PROGRAM AntiBlockingDamper
VAR
	fbHVACAntiBlockingDamper: FB_HVACAntiBlockingDamper;
	eDataSecurityType: E_HVACDataSecurityType := E_HVACDataSecurityType.eHVACDataSecurityType_Idle;
	bSetDefault: BOOL;
	bEnable: BOOL;
	bDisable: BOOL;
	ryDamper: REAL;
	dtSystemTime: DATE_AND_TIME;
	bReset: BOOL;
	eAntiBlockingMode: E_HVACAntiBlockingMode;
	iHoursDowntime: INT;
	iDayWeekly: INT;
	iHour: INT;
	iMinute: INT;
	iLenghtImpulse: INT;
	rQDamper: REAL;
	iQDamper: INT;
	bQAntiBlocking: BOOL;
	bInvalidParameter: BOOL;
END_VAR

fbHVACAntiBlockingDamper(
	eDataSecurityType:=eDataSecurityType, 
	bSetDefault:=bSetDefault, 
	bEnable:=bEnable, 
	bDisable:=bDisable, 
	ryDamper:=ryDamper, 
	dtSystemTime:=dtSystemTime, 
	bReset:=bReset, 
	eAntiBlockingMode:=eAntiBlockingMode, 
	iHoursDowntime:=iHoursDowntime, 
	iDayWeekly:=iDayWeekly, 
	iHour:=iHour, 
	iMinute:=iMinute, 
	iLenghtImpulse:=iLenghtImpulse, 
	rQDamper=>rQDamper, 
	iQDamper=>iQDamper, 
	bQAntiBlocking=>bQAntiBlocking, 
	bInvalidParameter=>bInvalidParameter);

END_PROGRAM

(* stored: Version 1.1.0.1, ProductVersion 3.1.4024.4
   POU AntiBlockingDamper: Id {e51c11cd-b3cd-4ad1-a243-7a29055f8b72}, SpecialFunc None *)
